// TIA Portal V17 export
// export: Created 2025-03-10T12:16:43.1890228Z, ExportSetting WithDefaults, DisplayName Totally Integrated Automation Portal, DisplayVersion V17 Update 8, DisplayName TIA Portal Openness, DisplayVersion V17 Update 8, DisplayName TIA Portal Version Control Interface, DisplayVersion V17, DisplayName SINAMICS Startdrive Advanced, DisplayVersion V17 SP2, DisplayName SINAMICS Startdrive G110M, G120, G120C, G120D, G120P, G115D, DisplayVersion V17 SP2, DisplayName SINAMICS Startdrive G130, G150, S120, S150, SINAMICS MV, S210, DisplayVersion V17 SP2, DisplayName STEP 7 Professional, DisplayVersion V17 Update 8, DisplayName SINUMERIK ONE STEP 7 Toolbox, DisplayVersion V17 Update 12, DisplayName SINUMERIK 840D sl STEP 7 Toolbox, DisplayVersion V17 Update 12, DisplayName STEP 7 Safety, DisplayVersion V17 Update 6, DisplayName WinCC Advanced, DisplayVersion V17 Update 8
FUNCTION "FC1090_IDEVICE_COM" : Void   // FC1090, LAD
{ S7_Optimized_Access := 'FALSE' }
AUTHOR : ETXETAR
VERSION : 1.0
// stored: AutoNumber false, IsIECCheckEnabled false, SetENOAutomatically false, UDAEnableTagReadback false
   VAR_TEMP
      COMMAND : Int;   // COMMAND
      BUSY : Bool;   // BUSY
   END_VAR
   VAR CONSTANT
      FC_NUMBER : Int := 1090;
   END_VAR
   VAR_TEMP   // added for the SCL form of the ladder/FBD networks
      _w1 : Bool;
   END_VAR
BEGIN

REGION Network 1: ACKNOWLEDGMENT FOR REINTEGRATION OF SEND DATA FOLLOWING COMMUNICAITON ERROR
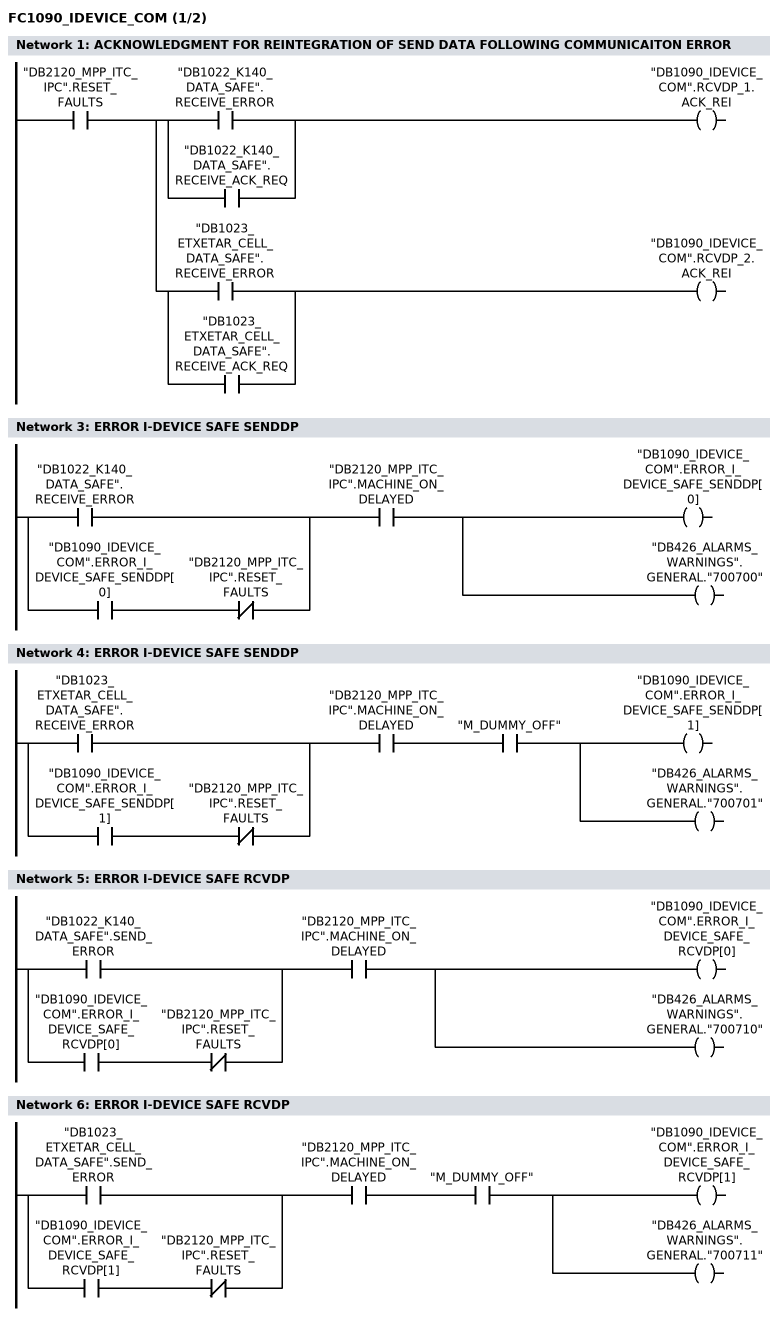
   RUNG wire#powerrail
      Contact( "DB2120_MPP_ITC_IPC".RESET_FAULTS )
      wire#w1
      Contact( "DB1022_K140_DATA_SAFE".RECEIVE_ERROR )
      wire#w2
      Coil( "DB1090_IDEVICE_COM".RCVDP_1.ACK_REI )
   END_RUNG
   RUNG wire#w1
      Contact( "DB1022_K140_DATA_SAFE".RECEIVE_ACK_REQ )
   END_RUNG wire#w2
   RUNG wire#w1
      Contact( "DB1023_ETXETAR_CELL_DATA_SAFE".RECEIVE_ERROR )
      wire#w3
      Coil( "DB1090_IDEVICE_COM".RCVDP_2.ACK_REI )
   END_RUNG
   RUNG wire#w1
      Contact( "DB1023_ETXETAR_CELL_DATA_SAFE".RECEIVE_ACK_REQ )
   END_RUNG wire#w3
   // the same network as SCL:
   "DB1090_IDEVICE_COM".RCVDP_1.ACK_REI := "DB2120_MPP_ITC_IPC".RESET_FAULTS AND ("DB1022_K140_DATA_SAFE".RECEIVE_ERROR OR "DB1022_K140_DATA_SAFE".RECEIVE_ACK_REQ);
   "DB1090_IDEVICE_COM".RCVDP_2.ACK_REI := "DB2120_MPP_ITC_IPC".RESET_FAULTS AND ("DB1023_ETXETAR_CELL_DATA_SAFE".RECEIVE_ERROR OR "DB1023_ETXETAR_CELL_DATA_SAFE".RECEIVE_ACK_REQ);
END_REGION

REGION Network 2: I-DEVICE SAFETY ALARMS
END_REGION

REGION Network 3: ERROR I-DEVICE SAFE SENDDP
   RUNG wire#powerrail
      Contact( "DB1022_K140_DATA_SAFE".RECEIVE_ERROR )
      wire#w1
      Contact( "DB2120_MPP_ITC_IPC".MACHINE_ON_DELAYED )
      wire#w2
      Coil( "DB1090_IDEVICE_COM".ERROR_I_DEVICE_SAFE_SENDDP[0] )
   END_RUNG
   RUNG wire#powerrail
      Contact( "DB1090_IDEVICE_COM".ERROR_I_DEVICE_SAFE_SENDDP[0] )
      I_Contact( "DB2120_MPP_ITC_IPC".RESET_FAULTS )
   END_RUNG wire#w1
   RUNG wire#w2
      Coil( "DB426_ALARMS_WARNINGS".GENERAL."700700" )
   END_RUNG
   // the same network as SCL:
   #_w1 := ("DB1022_K140_DATA_SAFE".RECEIVE_ERROR OR ("DB1090_IDEVICE_COM".ERROR_I_DEVICE_SAFE_SENDDP[0] AND NOT "DB2120_MPP_ITC_IPC".RESET_FAULTS)) AND "DB2120_MPP_ITC_IPC".MACHINE_ON_DELAYED;
   "DB1090_IDEVICE_COM".ERROR_I_DEVICE_SAFE_SENDDP[0] := ("DB1022_K140_DATA_SAFE".RECEIVE_ERROR OR ("DB1090_IDEVICE_COM".ERROR_I_DEVICE_SAFE_SENDDP[0] AND NOT "DB2120_MPP_ITC_IPC".RESET_FAULTS)) AND "DB2120_MPP_ITC_IPC".MACHINE_ON_DELAYED;
   "DB426_ALARMS_WARNINGS".GENERAL."700700" := #_w1;
END_REGION

REGION Network 4: ERROR I-DEVICE SAFE SENDDP
   RUNG wire#powerrail
      Contact( "DB1023_ETXETAR_CELL_DATA_SAFE".RECEIVE_ERROR )
      wire#w1
      Contact( "DB2120_MPP_ITC_IPC".MACHINE_ON_DELAYED )
      Contact( "M_DUMMY_OFF" )
      wire#w2
      Coil( "DB1090_IDEVICE_COM".ERROR_I_DEVICE_SAFE_SENDDP[1] )
   END_RUNG
   RUNG wire#powerrail
      Contact( "DB1090_IDEVICE_COM".ERROR_I_DEVICE_SAFE_SENDDP[1] )
      I_Contact( "DB2120_MPP_ITC_IPC".RESET_FAULTS )
   END_RUNG wire#w1
   RUNG wire#w2
      Coil( "DB426_ALARMS_WARNINGS".GENERAL."700701" )
   END_RUNG
   // the same network as SCL:
   #_w1 := ("DB1023_ETXETAR_CELL_DATA_SAFE".RECEIVE_ERROR OR ("DB1090_IDEVICE_COM".ERROR_I_DEVICE_SAFE_SENDDP[1] AND NOT "DB2120_MPP_ITC_IPC".RESET_FAULTS)) AND "DB2120_MPP_ITC_IPC".MACHINE_ON_DELAYED AND "M_DUMMY_OFF";
   "DB1090_IDEVICE_COM".ERROR_I_DEVICE_SAFE_SENDDP[1] := ("DB1023_ETXETAR_CELL_DATA_SAFE".RECEIVE_ERROR OR ("DB1090_IDEVICE_COM".ERROR_I_DEVICE_SAFE_SENDDP[1] AND NOT "DB2120_MPP_ITC_IPC".RESET_FAULTS)) AND "DB2120_MPP_ITC_IPC".MACHINE_ON_DELAYED AND "M_DUMMY_OFF";
   "DB426_ALARMS_WARNINGS".GENERAL."700701" := #_w1;
END_REGION

REGION Network 5: ERROR I-DEVICE SAFE RCVDP
   RUNG wire#powerrail
      Contact( "DB1022_K140_DATA_SAFE".SEND_ERROR )
      wire#w1
      Contact( "DB2120_MPP_ITC_IPC".MACHINE_ON_DELAYED )
      wire#w2
      Coil( "DB1090_IDEVICE_COM".ERROR_I_DEVICE_SAFE_RCVDP[0] )
   END_RUNG
   RUNG wire#powerrail
      Contact( "DB1090_IDEVICE_COM".ERROR_I_DEVICE_SAFE_RCVDP[0] )
      I_Contact( "DB2120_MPP_ITC_IPC".RESET_FAULTS )
   END_RUNG wire#w1
   RUNG wire#w2
      Coil( "DB426_ALARMS_WARNINGS".GENERAL."700710" )
   END_RUNG
   // the same network as SCL:
   #_w1 := ("DB1022_K140_DATA_SAFE".SEND_ERROR OR ("DB1090_IDEVICE_COM".ERROR_I_DEVICE_SAFE_RCVDP[0] AND NOT "DB2120_MPP_ITC_IPC".RESET_FAULTS)) AND "DB2120_MPP_ITC_IPC".MACHINE_ON_DELAYED;
   "DB1090_IDEVICE_COM".ERROR_I_DEVICE_SAFE_RCVDP[0] := ("DB1022_K140_DATA_SAFE".SEND_ERROR OR ("DB1090_IDEVICE_COM".ERROR_I_DEVICE_SAFE_RCVDP[0] AND NOT "DB2120_MPP_ITC_IPC".RESET_FAULTS)) AND "DB2120_MPP_ITC_IPC".MACHINE_ON_DELAYED;
   "DB426_ALARMS_WARNINGS".GENERAL."700710" := #_w1;
END_REGION

REGION Network 6: ERROR I-DEVICE SAFE RCVDP
   RUNG wire#powerrail
      Contact( "DB1023_ETXETAR_CELL_DATA_SAFE".SEND_ERROR )
      wire#w1
      Contact( "DB2120_MPP_ITC_IPC".MACHINE_ON_DELAYED )
      Contact( "M_DUMMY_OFF" )
      wire#w2
      Coil( "DB1090_IDEVICE_COM".ERROR_I_DEVICE_SAFE_RCVDP[1] )
   END_RUNG
   RUNG wire#powerrail
      Contact( "DB1090_IDEVICE_COM".ERROR_I_DEVICE_SAFE_RCVDP[1] )
      I_Contact( "DB2120_MPP_ITC_IPC".RESET_FAULTS )
   END_RUNG wire#w1
   RUNG wire#w2
      Coil( "DB426_ALARMS_WARNINGS".GENERAL."700711" )
   END_RUNG
   // the same network as SCL:
   #_w1 := ("DB1023_ETXETAR_CELL_DATA_SAFE".SEND_ERROR OR ("DB1090_IDEVICE_COM".ERROR_I_DEVICE_SAFE_RCVDP[1] AND NOT "DB2120_MPP_ITC_IPC".RESET_FAULTS)) AND "DB2120_MPP_ITC_IPC".MACHINE_ON_DELAYED AND "M_DUMMY_OFF";
   "DB1090_IDEVICE_COM".ERROR_I_DEVICE_SAFE_RCVDP[1] := ("DB1023_ETXETAR_CELL_DATA_SAFE".SEND_ERROR OR ("DB1090_IDEVICE_COM".ERROR_I_DEVICE_SAFE_RCVDP[1] AND NOT "DB2120_MPP_ITC_IPC".RESET_FAULTS)) AND "DB2120_MPP_ITC_IPC".MACHINE_ON_DELAYED AND "M_DUMMY_OFF";
   "DB426_ALARMS_WARNINGS".GENERAL."700711" := #_w1;
END_REGION

REGION Network 7: IMMEDIATE STOP ALARMS
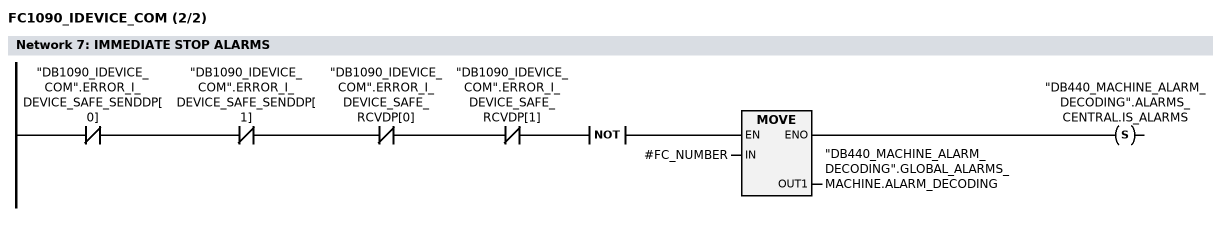
   RUNG wire#powerrail
      I_Contact( "DB1090_IDEVICE_COM".ERROR_I_DEVICE_SAFE_SENDDP[0] )
      I_Contact( "DB1090_IDEVICE_COM".ERROR_I_DEVICE_SAFE_SENDDP[1] )
      I_Contact( "DB1090_IDEVICE_COM".ERROR_I_DEVICE_SAFE_RCVDP[0] )
      I_Contact( "DB1090_IDEVICE_COM".ERROR_I_DEVICE_SAFE_RCVDP[1] )
      Not()
      { S7_GenerateENO := "TRUE" } Move(in := #FC_NUMBER, out1 => "DB440_MACHINE_ALARM_DECODING".GLOBAL_ALARMS_MACHINE.ALARM_DECODING)
      S_Coil( "DB440_MACHINE_ALARM_DECODING".ALARMS_CENTRAL.IS_ALARMS )
   END_RUNG
   // the same network as SCL:
   // ENO of a box is taken as its EN; it also drops when the box reports an error
   IF NOT (NOT "DB1090_IDEVICE_COM".ERROR_I_DEVICE_SAFE_SENDDP[0] AND NOT "DB1090_IDEVICE_COM".ERROR_I_DEVICE_SAFE_SENDDP[1] AND NOT "DB1090_IDEVICE_COM".ERROR_I_DEVICE_SAFE_RCVDP[0] AND NOT "DB1090_IDEVICE_COM".ERROR_I_DEVICE_SAFE_RCVDP[1]) THEN
       "DB440_MACHINE_ALARM_DECODING".GLOBAL_ALARMS_MACHINE.ALARM_DECODING := #FC_NUMBER;
       "DB440_MACHINE_ALARM_DECODING".ALARMS_CENTRAL.IS_ALARMS := TRUE;
   END_IF;
END_REGION
END_FUNCTION
